// Mitsubishi GX Works2 project: v1_final   PLC: Q02/Q02H

PROGRAM MAIN
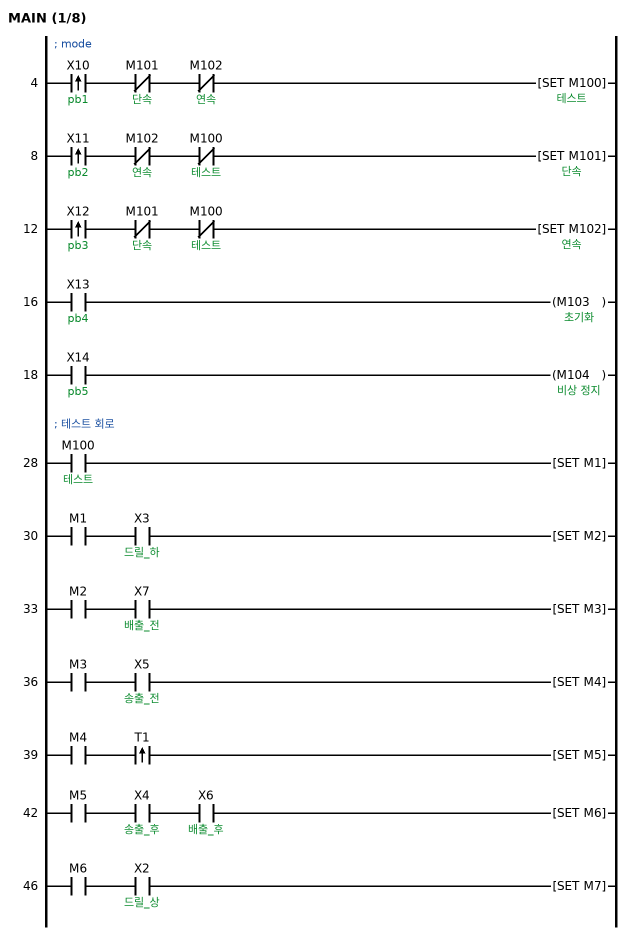
; mode
4     LDP     X10  ; pb1
      ANI     M101  ; 단속
      ANI     M102  ; 연속
      SET     M100  ; 테스트
8     LDP     X11  ; pb2
      ANI     M102  ; 연속
      ANI     M100  ; 테스트
      SET     M101  ; 단속
12    LDP     X12  ; pb3
      ANI     M101  ; 단속
      ANI     M100  ; 테스트
      SET     M102  ; 연속
16    LD      X13  ; pb4
      OUT     M103  ; 초기화
18    LD      X14  ; pb5
      OUT     M104  ; 비상 정지
; 테스트 회로
28    LD      M100  ; 테스트
      SET     M1
30    LD      M1
      AND     X3  ; 드릴_하
      SET     M2
33    LD      M2
      AND     X7  ; 배출_전
      SET     M3
36    LD      M3
      AND     X5  ; 송출_전
      SET     M4
39    LD      M4
      ANDP    T1
      SET     M5
42    LD      M5
      AND     X4  ; 송출_후
      AND     X6  ; 배출_후
      SET     M6
46    LD      M6
      AND     X2  ; 드릴_상
      SET     M7
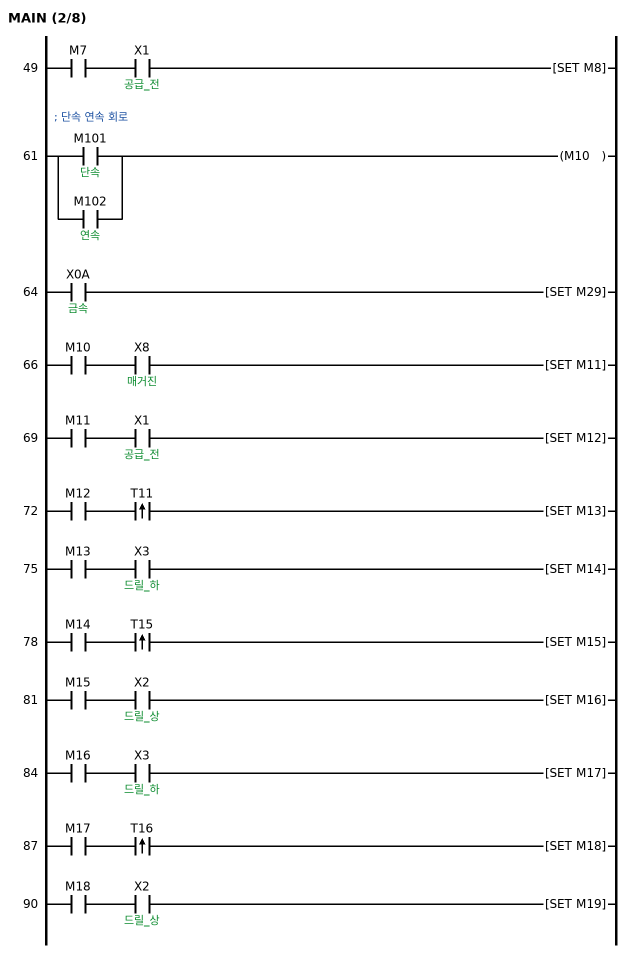
49    LD      M7
      AND     X1  ; 공급_전
      SET     M8
; 단속 연속 회로
61    LD      M101  ; 단속
      OR      M102  ; 연속
      OUT     M10
64    LD      X0A  ; 금속
      SET     M29
66    LD      M10
      AND     X8  ; 매거진
      SET     M11
69    LD      M11
      AND     X1  ; 공급_전
      SET     M12
72    LD      M12
      ANDP    T11
      SET     M13
75    LD      M13
      AND     X3  ; 드릴_하
      SET     M14
78    LD      M14
      ANDP    T15
      SET     M15
81    LD      M15
      AND     X2  ; 드릴_상
      SET     M16
84    LD      M16
      AND     X3  ; 드릴_하
      SET     M17
87    LD      M17
      ANDP    T16
      SET     M18
90    LD      M18
      AND     X2  ; 드릴_상
      SET     M19
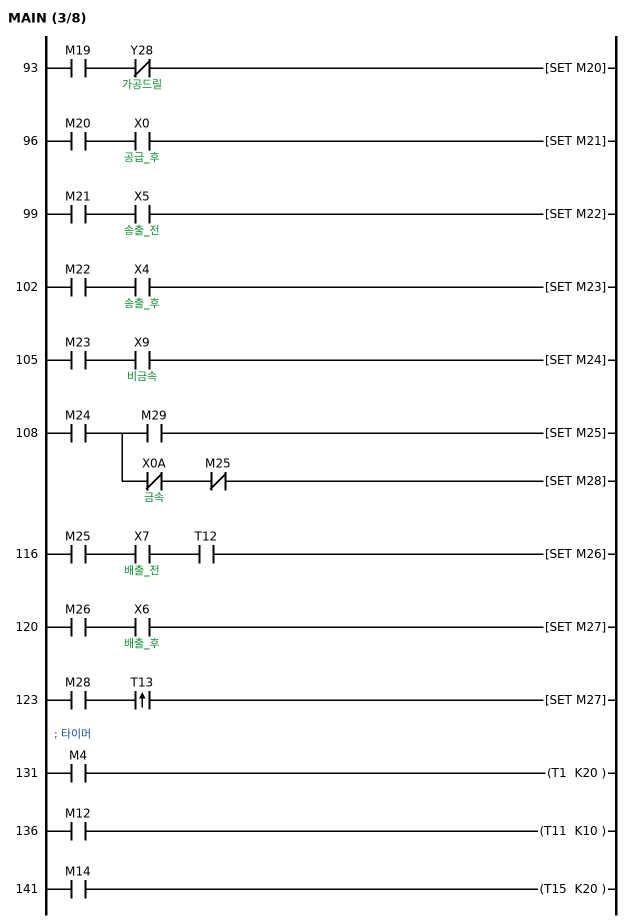
93    LD      M19
      ANI     Y28  ; 가공드릴
      SET     M20
96    LD      M20
      AND     X0  ; 공급_후
      SET     M21
99    LD      M21
      AND     X5  ; 송출_전
      SET     M22
102   LD      M22
      AND     X4  ; 송출_후
      SET     M23
105   LD      M23
      AND     X9  ; 비금속
      SET     M24
108   LD      M24
      MPS
      AND     M29
      SET     M25
      MPP
      ANI     X0A  ; 금속
      ANI     M25
      SET     M28
116   LD      M25
      AND     X7  ; 배출_전
      AND     T12
      SET     M26
120   LD      M26
      AND     X6  ; 배출_후
      SET     M27
123   LD      M28
      ANDP    T13
      SET     M27
; 타이머
131   LD      M4
      OUT     T1 K20
136   LD      M12
      OUT     T11 K10
141   LD      M14
      OUT     T15 K20
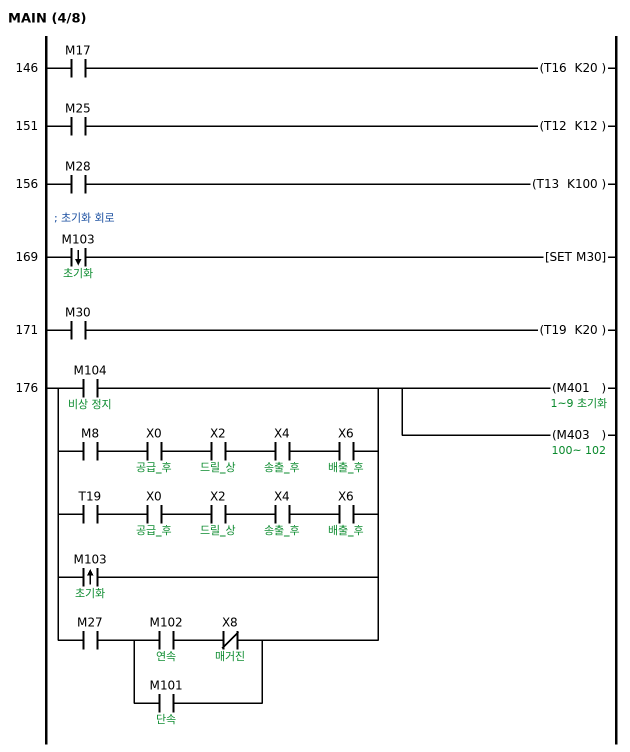
146   LD      M17
      OUT     T16 K20
151   LD      M25
      OUT     T12 K12
156   LD      M28
      OUT     T13 K100
; 초기화 회로
169   LDF     M103  ; 초기화
      SET     M30
171   LD      M30
      OUT     T19 K20
176   LD      M104  ; 비상 정지
      LD      M8
      AND     X0  ; 공급_후
      AND     X2  ; 드릴_상
      AND     X4  ; 송출_후
      AND     X6  ; 배출_후
      ORB
      LD      T19
      AND     X0  ; 공급_후
      AND     X2  ; 드릴_상
      AND     X4  ; 송출_후
      AND     X6  ; 배출_후
      ORB
      ORP     M103  ; 초기화
      LD      M27
      LD      M102  ; 연속
      ANI     X8  ; 매거진
      OR      M101  ; 단속
      ANB
      ORB
      OUT     M401  ; 1~9 초기화
      OUT     M403  ; 100~ 102
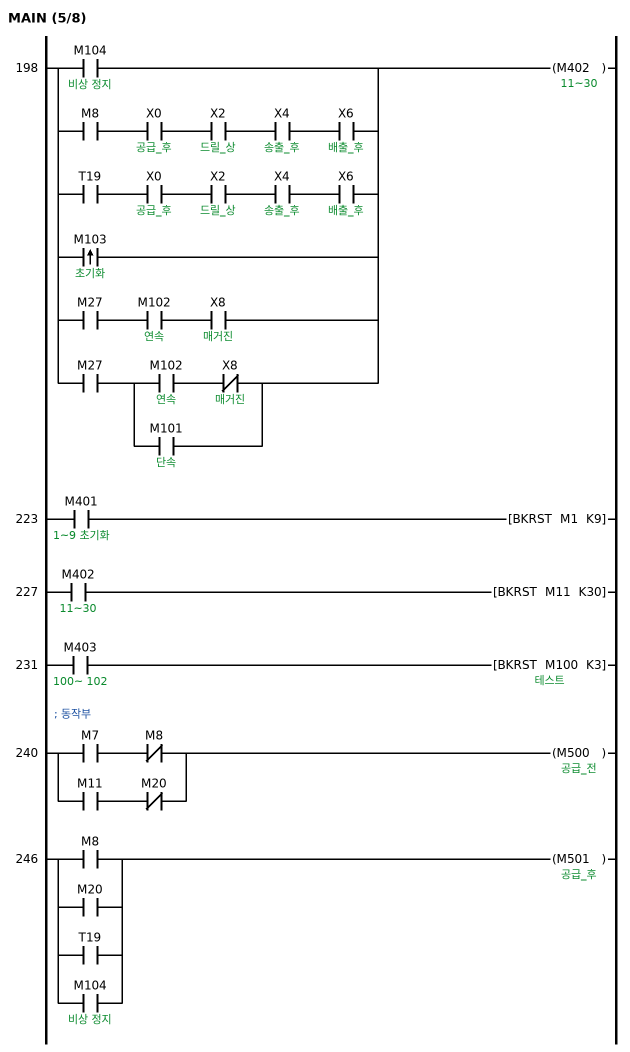
198   LD      M104  ; 비상 정지
      LD      M8
      AND     X0  ; 공급_후
      AND     X2  ; 드릴_상
      AND     X4  ; 송출_후
      AND     X6  ; 배출_후
      ORB
      LD      T19
      AND     X0  ; 공급_후
      AND     X2  ; 드릴_상
      AND     X4  ; 송출_후
      AND     X6  ; 배출_후
      ORB
      ORP     M103  ; 초기화
      LD      M27
      AND     M102  ; 연속
      AND     X8  ; 매거진
      ORB
      LD      M27
      LD      M102  ; 연속
      ANI     X8  ; 매거진
      OR      M101  ; 단속
      ANB
      ORB
      OUT     M402  ; 11~30
223   LD      M401  ; 1~9 초기화
      BKRST   M1 K9
227   LD      M402  ; 11~30
      BKRST   M11 K30
231   LD      M403  ; 100~ 102
      BKRST   M100 K3
; 동작부
240   LD      M7
      ANI     M8
      LD      M11
      ANI     M20
      ORB
      OUT     M500  ; 공급_전
246   LD      M8
      OR      M20
      OR      T19
      OR      M104  ; 비상 정지
      OUT     M501  ; 공급_후
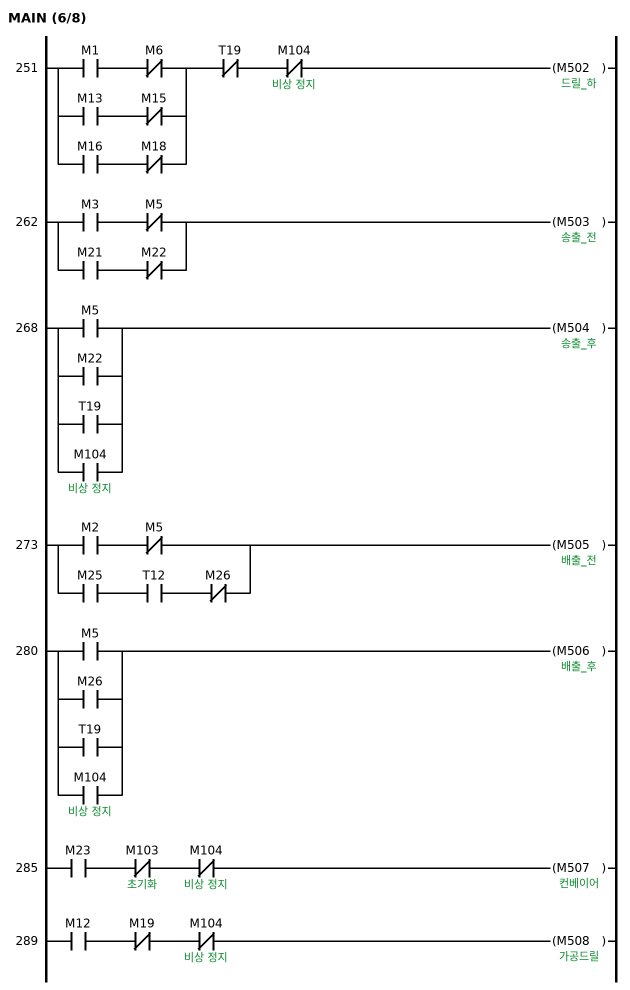
251   LD      M1
      ANI     M6
      LD      M13
      ANI     M15
      ORB
      LD      M16
      ANI     M18
      ORB
      ANI     T19
      ANI     M104  ; 비상 정지
      OUT     M502  ; 드릴_하
262   LD      M3
      ANI     M5
      LD      M21
      ANI     M22
      ORB
      OUT     M503  ; 송출_전
268   LD      M5
      OR      M22
      OR      T19
      OR      M104  ; 비상 정지
      OUT     M504  ; 송출_후
273   LD      M2
      ANI     M5
      LD      M25
      AND     T12
      ANI     M26
      ORB
      OUT     M505  ; 배출_전
280   LD      M5
      OR      M26
      OR      T19
      OR      M104  ; 비상 정지
      OUT     M506  ; 배출_후
285   LD      M23
      ANI     M103  ; 초기화
      ANI     M104  ; 비상 정지
      OUT     M507  ; 컨베이어
289   LD      M12
      ANI     M19
      ANI     M104  ; 비상 정지
      OUT     M508  ; 가공드릴
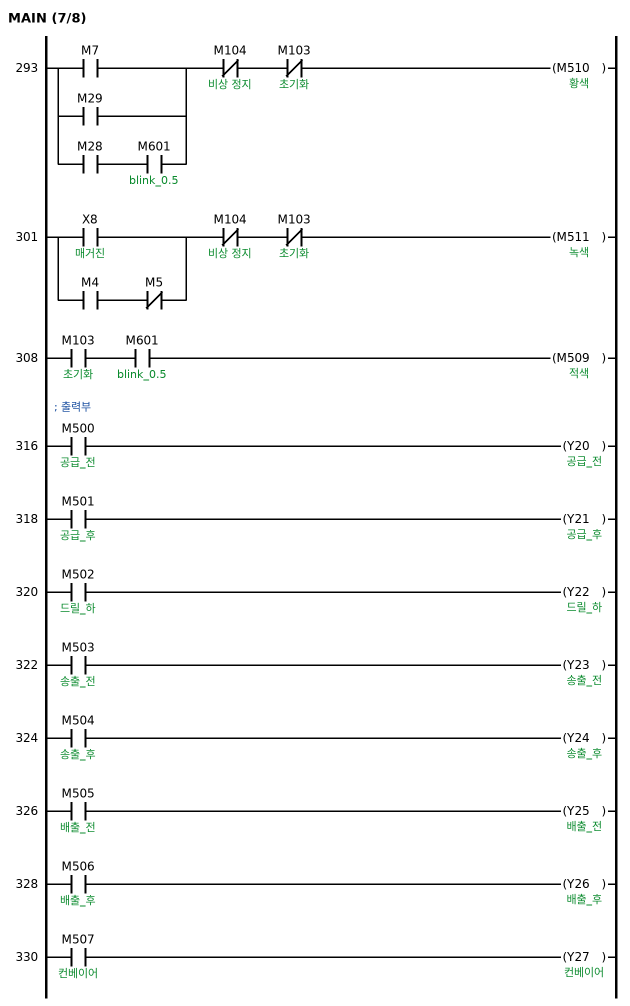
293   LD      M7
      OR      M29
      LD      M28
      AND     M601  ; blink_0.5
      ORB
      ANI     M104  ; 비상 정지
      ANI     M103  ; 초기화
      OUT     M510  ; 황색
301   LD      X8  ; 매거진
      LD      M4
      ANI     M5
      ORB
      ANI     M104  ; 비상 정지
      ANI     M103  ; 초기화
      OUT     M511  ; 녹색
308   LD      M103  ; 초기화
      AND     M601  ; blink_0.5
      OUT     M509  ; 적색
; 출력부
316   LD      M500  ; 공급_전
      OUT     Y20  ; 공급_전
318   LD      M501  ; 공급_후
      OUT     Y21  ; 공급_후
320   LD      M502  ; 드릴_하
      OUT     Y22  ; 드릴_하
322   LD      M503  ; 송출_전
      OUT     Y23  ; 송출_전
324   LD      M504  ; 송출_후
      OUT     Y24  ; 송출_후
326   LD      M505  ; 배출_전
      OUT     Y25  ; 배출_전
328   LD      M506  ; 배출_후
      OUT     Y26  ; 배출_후
330   LD      M507  ; 컨베이어
      OUT     Y27  ; 컨베이어
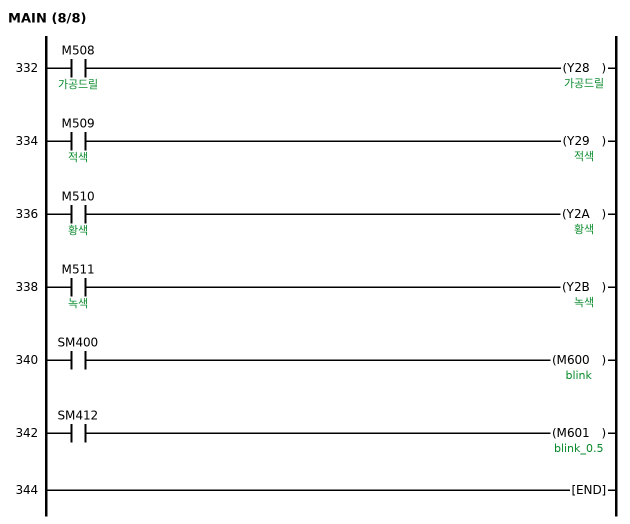
332   LD      M508  ; 가공드릴
      OUT     Y28  ; 가공드릴
334   LD      M509  ; 적색
      OUT     Y29  ; 적색
336   LD      M510  ; 황색
      OUT     Y2A  ; 황색
338   LD      M511  ; 녹색
      OUT     Y2B  ; 녹색
340   LD      SM400
      OUT     M600  ; blink
342   LD      SM412
      OUT     M601  ; blink_0.5
344   END
END_PROGRAM

PROGRAM MAIN1
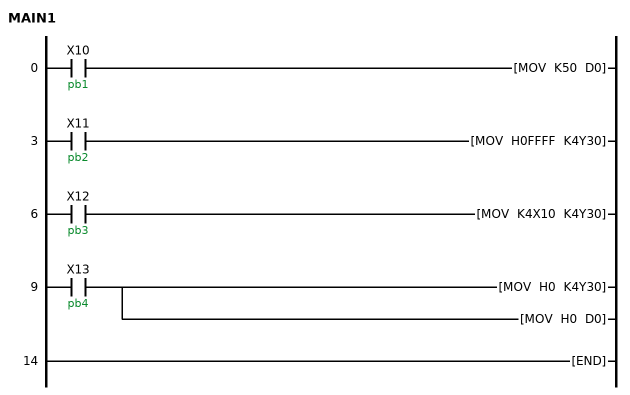
0     LD      X10  ; pb1
      MOV     K50 D0
3     LD      X11  ; pb2
      MOV     H0FFFF K4Y30
6     LD      X12  ; pb3
      MOV     K4X10 K4Y30
9     LD      X13  ; pb4
      MOV     H0 K4Y30
      MOV     H0 D0
14    END
END_PROGRAM

PROGRAM MAIN2
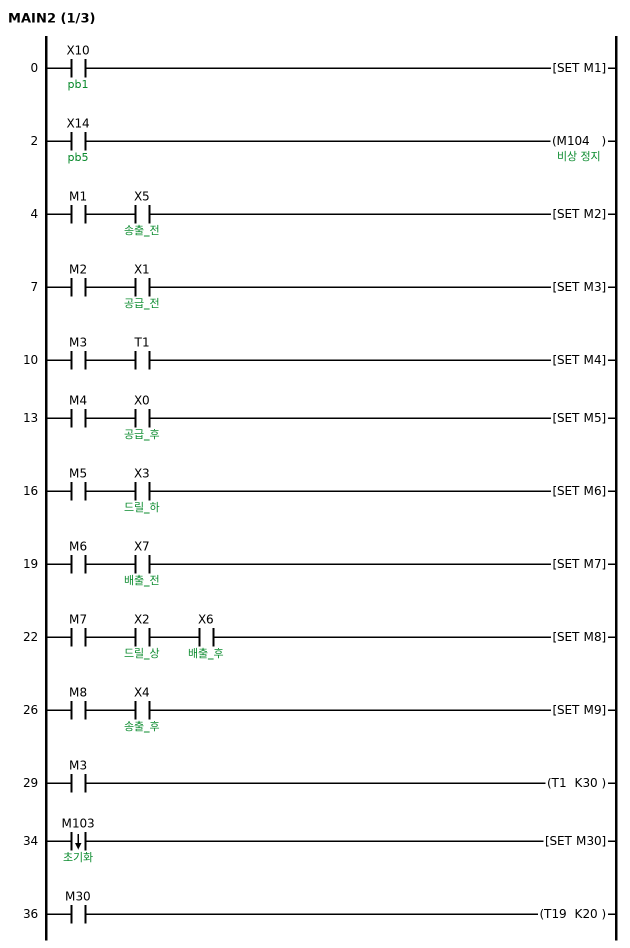
0     LD      X10  ; pb1
      SET     M1
2     LD      X14  ; pb5
      OUT     M104  ; 비상 정지
4     LD      M1
      AND     X5  ; 송출_전
      SET     M2
7     LD      M2
      AND     X1  ; 공급_전
      SET     M3
10    LD      M3
      AND     T1
      SET     M4
13    LD      M4
      AND     X0  ; 공급_후
      SET     M5
16    LD      M5
      AND     X3  ; 드릴_하
      SET     M6
19    LD      M6
      AND     X7  ; 배출_전
      SET     M7
22    LD      M7
      AND     X2  ; 드릴_상
      AND     X6  ; 배출_후
      SET     M8
26    LD      M8
      AND     X4  ; 송출_후
      SET     M9
29    LD      M3
      OUT     T1 K30
34    LDF     M103  ; 초기화
      SET     M30
36    LD      M30
      OUT     T19 K20
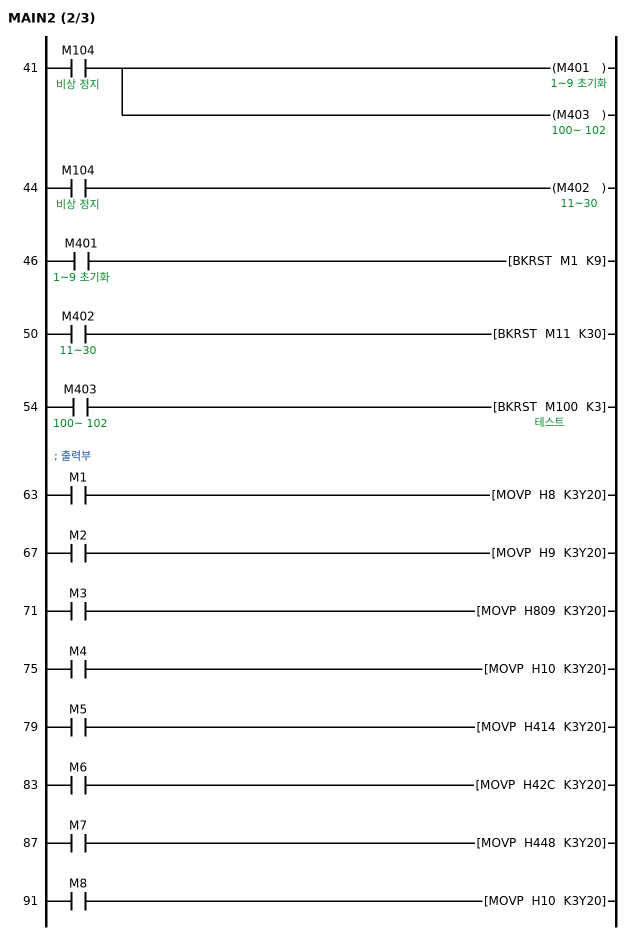
41    LD      M104  ; 비상 정지
      OUT     M401  ; 1~9 초기화
      OUT     M403  ; 100~ 102
44    LD      M104  ; 비상 정지
      OUT     M402  ; 11~30
46    LD      M401  ; 1~9 초기화
      BKRST   M1 K9
50    LD      M402  ; 11~30
      BKRST   M11 K30
54    LD      M403  ; 100~ 102
      BKRST   M100 K3  ; 테스트
; 출력부
63    LD      M1
      MOVP    H8 K3Y20  ; 공급_전
67    LD      M2
      MOVP    H9 K3Y20
71    LD      M3
      MOVP    H809 K3Y20
75    LD      M4
      MOVP    H10 K3Y20
79    LD      M5
      MOVP    H414 K3Y20
83    LD      M6
      MOVP    H42C K3Y20
87    LD      M7
      MOVP    H448 K3Y20
91    LD      M8
      MOVP    H10 K3Y20
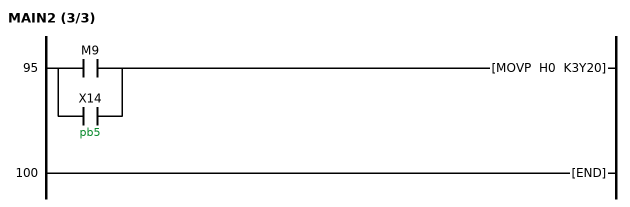
95    LD      M9
      OR      X14  ; pb5
      MOVP    H0 K3Y20
100   END
END_PROGRAM

// device comments not shown above
M400  ; 비상 타이머
